FUNCTION_BLOCK SkidMagazine EXTENDS MaterialHolder
VAR_OUTPUT
	inPosition AT %I* : ARRAY[1..2] OF BOOL;
END_VAR

SUPER^();

METHOD setOccupancy : BOOL
VAR_INPUT
	i : INT;
	occupancy : BOOL;
END_VAR
VAR_OUTPUT
	errorBounds : BOOL;
END_VAR
errorBounds := i < LOWER_BOUND(slots, 1) OR i > UPPER_BOUND(slots, 1);

IF NOT errorBounds THEN
	occupied[i] := occupancy;
END_IF

IF hmiTable <> 0 THEN
	writeHmiTable();
END_IF
END_METHOD

END_FUNCTION_BLOCK

(* stored: Version 1.1.0.1, ProductVersion 3.1.4024.11
   POU SkidMagazine: Id {cc4e8e9a-d375-4787-b88d-f0c2dcecd871}, SpecialFunc None
   Method setOccupancy: Id {30a7aa2b-716c-4159-99e8-4869a1f9802b} *)
